// TwinCAT 3 PLC project Untitled2
// ProgramVersion: 3.1.4023.0
// libraries:
//   Tc2_Standard, * (Beckhoff Automation GmbH)
//   Tc2_System, * (Beckhoff Automation GmbH)
//   Tc2_TcpIp, * (Beckhoff Automation GmbH)
//   Tc3_Module, * (Beckhoff Automation GmbH)
// project tree:
//   GVLs/ GVL.TcGVL
//   / PlcTask.TcTTO
//   POUs/ MAIN.TcPOU
// real-time tasks:
//   TASK PlcTask1: cycle T#10ms, priority 21, ADS port 351
//   TASK Task 3: cycle T#1ms, priority 1, ADS port 301
// I/O:
//   DEVICE Device 1 (TC3 EIP Adapter), AmsNetId 5.104.86.109.2.1
//     Beckhoff CX8190 EIP EDS Test
// variable links:
//   Untitled2/Untitled2 Instance <-> Device 1 (TC3 EIP Adapter)/Beckhoff CX8190 EIP EDS Test
//     PlcTask Inputs/GVL.Output_100 <-> Assembly 1 (Input/Output)/Inputs/Input_100
//     PlcTask Outputs/GVL.Input_100 <-> Assembly 1 (Input/Output)/Outputs/Output_100

CONFIGURATION Untitled2
    RESOURCE PLC ON TwinCAT3
        TASK PlcTask(INTERVAL := T#10ms, PRIORITY := 21);
        PROGRAM MAIN WITH PlcTask : MAIN;
    END_RESOURCE
END_CONFIGURATION

// ---- GVLs/GVL.TcGVL
{attribute 'qualified_only'}
VAR_GLOBAL
	
	Output_100 AT %i*: ARRAY[0..100] OF Byte;
	Input_100 AT %Q*: ARRAY[0..100] OF Byte;
END_VAR

// ---- POUs/MAIN.TcPOU
PROGRAM MAIN
VAR
END_VAR

END_PROGRAM
